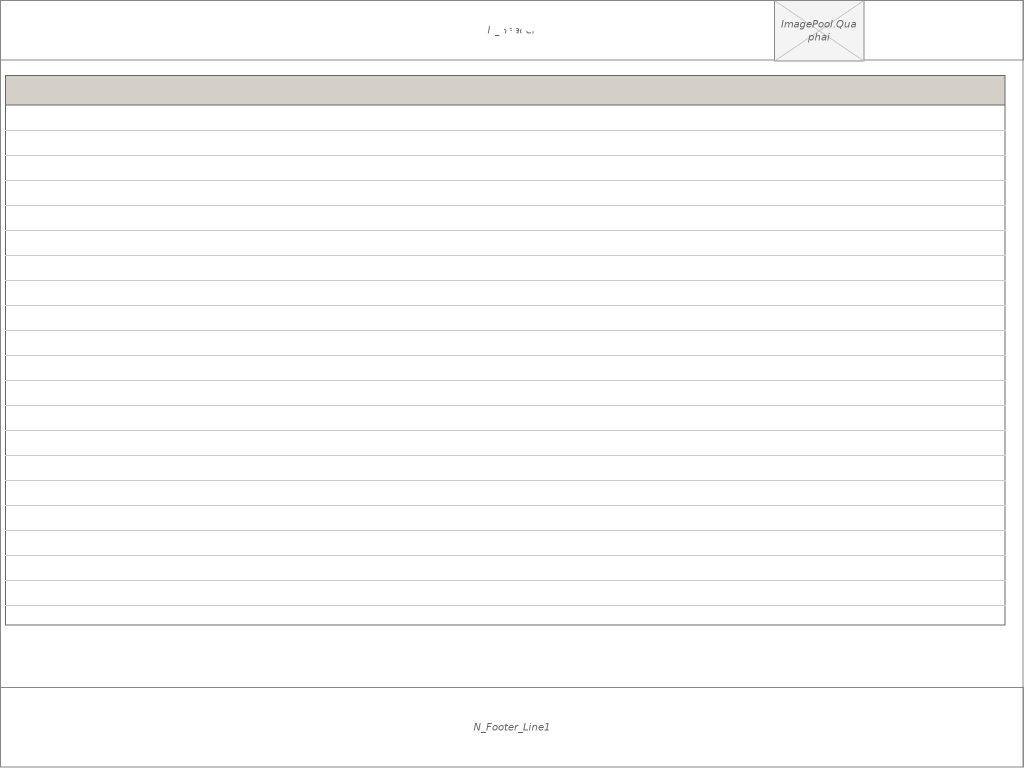
VISUALIZATION N_Alarm  // 1024x768
    Table (5,75 1000x550), invisible if: Not bVN, data array: AlarmList
        p3854506369: AlarmList[1,INDEX]
        p1892666644: AlarmList[2,INDEX]
        p338671338: AlarmList[3,INDEX]
        p2170511999: AlarmList[4,INDEX]
        p511219082: Mô tả
        p1755163831: Trạng thái
        p4092479075: Thời gian
    Table (5,75 1000x550), invisible if: bVN, data array: AlarmList3
        p3854506369: AlarmList3[1,INDEX]
        p1892666644: AlarmList3[2,INDEX]
        p338671338: AlarmList[3,INDEX]
        p2170511999: AlarmList[4,INDEX]
        p511219082: Describe
        p1755163831: Status
        p4092479075: Time
        p1791247317: AlarmList3[3,INDEX]
        p262371475: AlarmList3[4,INDEX]
    Frame (0,687 1024x80)
        shows N_Footer_Line1()
    Frame (0,0 1024x60)
        shows N_Header()
    Textfield (353,5 400x50), "MÀN HÌNH LỖI TRẠM 1"
    Image (774,0 90x61), image: ImagePool.Qua phai
        OnMouseClick: change screen: N_Alarm_1
END_VISUALIZATION

(* stored: Version 1.1.0.1, ProductVersion 3.1.4024.12
   Visu N_Alarm: Id {ddcc1c04-d230-473a-b577-0e588c000c6d} *)
